{attribute 'qualified_only'}
{attribute 'strict'}
{attribute 'to_string'}
TYPE E_Alarm :
(
	AL000,
	AL001,
	AL002,
	AL003,
	AL004,
	AL005,
	AL006,
	AL007,
	AL008,
	AL009,
	AL010,
	AL011,
	AL012,
	AL013,
	AL014,
	AL015,
	AL016,
	AL017,
	AL018,
	AL019,
	AL020,
	AL021,
	AL022,
	AL023,
	AL024,
	AL025,
	AL026,
	AL027,
	AL028,
	AL029,
	AL030,
	AL031,
	AL032,
	AL033,
	AL034,
	AL035,
	AL036,
	AL037,
	AL038,
	AL039,
	AL040,
	AL041,
	AL042,
	AL043,
	AL044,
	AL045,
	AL046,
	AL047,
	AL048,
	AL049,
	AL050,
	AL051,
	AL052,
	AL053,
	AL054,
	AL055,
	AL056,
	AL057,
	AL058,
	AL059,
	AL060,
	AL061,
	AL062,
	AL063,
	AL064,
	AL065,
	AL066,
	AL067,
	AL068,
	AL069,
	AL070,
	AL071,
	AL072,
	AL073,
	AL074,
	AL075,
	AL076,
	AL077,
	AL078,
	AL079,
	AL080,
	AL081,
	AL082,
	AL083,
	AL084,
	AL085,
	AL086,
	AL087,
	AL088,
	AL089,
	AL090,
	AL091,
	AL092,
	AL093,
	AL094,
	AL095,
	AL096,
	AL097,
	AL098,
	AL099,
	AL100,
	AL101,
	AL102,
	AL103,
	AL104,
	AL105,
	AL106,
	AL107,
	AL108,
	AL109,
	AL110,
	AL111,
	AL112,
	AL113,
	AL114,
	AL115,
	AL116,
	AL117,
	AL118,
	AL119,
	AL120,
	AL121,
	AL122,
	AL123,
	AL124,
	AL125,
	AL126,
	AL127,
	AL128,
	AL129,
	AL130,
	AL131,
	AL132,
	AL133,
	AL134,
	AL135,
	AL136,
	AL137,
	AL138,
	AL139,
	AL140,
	AL141,
	AL142,
	AL143,
	AL144,
	AL145,
	AL146,
	AL147,
	AL148,
	AL149,
	AL150,
	AL151,
	AL152,
	AL153,
	AL154,
	AL155,
	AL156,
	AL157,
	AL158,
	AL159,
	AL160,
	AL161,
	AL162,
	AL163,
	AL164,
	AL165,
	AL166,
	AL167,
	AL168,
	AL169,
	AL170,
	AL171,
	AL172,
	AL173,
	AL174,
	AL175,
	AL176,
	AL177,
	AL178,
	AL179,
	AL180,
	AL181,
	AL182,
	AL183,
	AL184,
	AL185,
	AL186,
	AL187,
	AL188,
	AL189,
	AL190,
	AL191,
	AL192,
	AL193,
	AL194,
	AL195,
	AL196,
	AL197,
	AL198,
	AL199,
	AL200,
	AL201,
	AL202,
	AL203,
	AL204,
	AL205,
	AL206,
	AL207,
	AL208,
	AL209,
	AL210,
	AL211,
	AL212,
	AL213,
	AL214,
	AL215,
	AL216,
	AL217,
	AL218,
	AL219,
	AL220,
	AL221,
	AL222,
	AL223,
	AL224,
	AL225,
	AL226,
	AL227,
	AL228,
	AL229,
	AL230,
	AL231,
	AL232,
	AL233,
	AL234,
	AL235,
	AL236,
	AL237,
	AL238,
	AL239,
	AL240,
	AL241,
	AL242,
	AL243,
	AL244,
	AL245,
	AL246,
	AL247,
	AL248,
	AL249,
	AL250,
	AL251,
	AL252,
	AL253,
	AL254,
	AL255,
	AL256,
	AL257,
	AL258,
	AL259,
	AL260,
	AL261,
	AL262,
	AL263,
	AL264,
	AL265,
	AL266,
	AL267,
	AL268,
	AL269,
	AL270,
	AL271,
	AL272,
	AL273,
	AL274,
	AL275,
	AL276,
	AL277,
	AL278,
	AL279,
	AL280,
	AL281,
	AL282,
	AL283,
	AL284,
	AL285,
	AL286,
	AL287,
	AL288,
	AL289,
	AL290,
	AL291,
	AL292,
	AL293,
	AL294,
	AL295,
	AL296,
	AL297,
	AL298,
	AL299,
	AL300,
	AL301,
	AL302,
	AL303,
	AL304,
	AL305,
	AL306,
	AL307,
	AL308,
	AL309,
	AL310,
	AL311,
	AL312,
	AL313,
	AL314,
	AL315,
	AL316,
	AL317,
	AL318,
	AL319,
	AL320,
	AL321,
	AL322,
	AL323,
	AL324,
	AL325,
	AL326,
	AL327,
	AL328,
	AL329,
	AL330,
	AL331,
	AL332,
	AL333,
	AL334,
	AL335,
	AL336,
	AL337,
	AL338,
	AL339,
	AL340,
	AL341,
	AL342,
	AL343,
	AL344,
	AL345,
	AL346,
	AL347,
	AL348,
	AL349,
	AL350,
	AL351,
	AL352,
	AL353,
	AL354,
	AL355,
	AL356,
	AL357,
	AL358,
	AL359,
	AL360,
	AL361,
	AL362,
	AL363,
	AL364,
	AL365,
	AL366,
	AL367,
	AL368,
	AL369,
	AL370,
	AL371,
	AL372,
	AL373,
	AL374,
	AL375,
	AL376,
	AL377,
	AL378,
	AL379,
	AL380,
	AL381,
	AL382,  
	AL383,
	AL384,
	AL385,
	AL386,
	AL387,
	AL388,
	AL389,  
	AL390,
	AL391,
	AL392,
	AL393,
	AL394,
	AL395,
	AL396,
	AL397,
	AL398,
	AL399,
	AL400,//B槽主軸伺服馬達_軸錯誤異常   
	AL401,//B槽清洗內罩升降1馬達_軸錯誤異常
	AL402,//B槽清洗內罩升降2馬達_軸錯誤異常
	AL403,//B槽清洗外罩升降1馬達_軸錯誤異常
	AL404,//B槽清洗外罩升降2馬達_軸錯誤異常
	AL405,//B槽噴頭擺臂升降馬達_軸錯誤異常 
	AL406,//B槽噴頭擺臂馬達_軸錯誤異常   
	AL407,//B槽頂PIN升降馬達_軸錯誤異常
	AL408,//B槽噴頭X軸馬達_軸錯誤異常   
	AL409,//B槽噴頭Y1軸馬達_軸錯誤異常  
	AL410,//B槽噴頭Y2軸馬達_軸錯誤異常  
	AL411,//B槽噴頭Z軸馬達_軸錯誤異常
	AL412,//B槽噴頭T軸馬達_軸錯誤異常 
	AL413,//B槽主軸伺服馬達_驅動器異常   
	AL414,//B槽清洗內罩升降1馬達_驅動器異常
	AL415,//B槽清洗內罩升降2馬達_驅動器異常
	AL416,//B槽清洗外罩升降1馬達_驅動器異常
	AL417,//B槽清洗外罩升降2馬達_驅動器異常
	AL418,//B槽噴頭擺臂升降馬達_驅動器異常 
	AL419,//B槽噴頭擺臂馬達_驅動器異常   
	AL420,//B槽頂PIN升降馬達_驅動器異常 
	AL421,//B槽噴頭X軸馬達_驅動器異常   
	AL422,//B槽噴頭Y1軸馬達_驅動器異常  
	AL423,//B槽噴頭Y2軸馬達_驅動器異常  
	AL424,//B槽噴頭Z軸馬達_驅動器異常   
	AL425,//B槽噴頭T軸馬達_驅動器異常   
	AL426,//                 
	AL427,//                 
	AL428,//                 
	AL429,//                 
	AL430,//清洗內罩升降1到位檢知異常    
	AL431,//清洗內罩升降2到位檢知異常    
	AL432,//清洗外罩升降1到位檢知異常    
	AL433,//清洗外罩升降2到位檢知異常    
	AL434,//噴頭X軸到位檢知異常       
	AL435,//噴頭Z軸到位檢知異常       
	AL436,//噴頭Y1軸到位檢知異常      
	AL437,//噴頭Y2軸到位檢知異常      
	AL438,//頂PIN升降到位檢知異常     
	AL439,//噴頭擺臂升降到位檢知異常     
	AL440,//噴頭擺臂擺動到位檢知異常     
	AL441,//閘門磁簧開關1(關)異常     
	AL442,//閘門磁簧開關1(開)異常     
	AL443,//閘門磁簧開關2(關)異常     
	AL444,//閘門磁簧開關2(開)異常     
	AL445,//上擺臂定位汽缸磁簧開關(定位)異常
	AL446,//上擺臂定位汽缸磁簧開關(退)異常 
	AL447,//下擺臂定位汽缸磁簧開關(定位)異常
	AL448,//下擺臂定位汽缸磁簧開關(退)異常 
	AL449,//上擺臂切換光電素子異常      
	AL450,//下擺臂切換光電素子異常      
	AL451,//DIW混CO2加熱器EGO異常  
	AL452,//DIW加熱器EGO異常      
	AL453,//漏液檢知器異常          
	AL454,//                 
	AL455,//                 
	AL456,//                 
	AL457,//                 
	AL458,//                 
	AL459,//                 
	AL460,//                 
	AL461,//                 
	AL462,//                 
	AL463,//                 
	AL464,//                 
	AL465,//                 
	AL466,//                 
	AL467,//                 
	AL468,//                 
	AL469,//                 
	AL470,//                 
	AL471,//                 
	AL472,//                 
	AL473,//                 
	AL474,//                 
	AL475,//                 
	AL476,//                 
	AL477,//                 
	AL478,//                 
	AL479,//                 
	AL480,//                 
	AL481,//                 
	AL482,//                 
	AL483,//                 
	AL484,//                 
	AL485,//                 
	AL486,//                 
	AL487,//                 
	AL488,//                 
	AL489,//                 
	AL490,//                 
	AL491,//                 
	AL492,//                 
	AL493,//                 
	AL494,//                 
	AL495,//                 
	AL496,//                 
	AL497,//                 
	AL498,//                 
	AL499,//                 
	AL500,//                 
	AL501,//                 
	AL502,//                 
	AL503,//                 
	AL504,//                 
	AL505,//                 
	AL506,//                 
	AL507,//                 
	AL508,//                 
	AL509,//                 
	AL510,//                 
	AL511,//                 
	AL512,//                 
	AL513,//                 
	AL514,//                 
	AL515,//                 
	AL516,//                 
	AL517,//                 
	AL518,//                 
	AL519,//                 
	AL520,//                 
	AL521,//                 
	AL522,//                 
	AL523,//                 
	AL524,//                 
	AL525,//                 
	AL526,//                 
	AL527,//                 
	AL528,//                 
	AL529,//                 
	AL530,//                 
	AL531,//                 
	AL532,//                 
	AL533,//                 
	AL534,//                 
	AL535,//                 
	AL536,//                 
	AL537,//                 
	AL538,//                 
	AL539,//                 
	AL540,//                 
	AL541,//                 
	AL542,//                 
	AL543,//                 
	AL544,//                 
	AL545,//                 
	AL546,//                 
	AL547,//                 
	AL548,//                 
	AL549,//                 
	AL550,//                 
	AL551,//                 
	AL552,//                 
	AL553,//                 
	AL554,//                 
	AL555,//                 
	AL556,//                 
	AL557,//                 
	AL558,//                 
	AL559,//                 
	AL560,//                 
	AL561,//                 
	AL562,//                 
	AL563,//                 
	AL564,//                 
	AL565,//                 
	AL566,//                 
	AL567,//                 
	AL568,//                 
	AL569,//                 
	AL570,//                 
	AL571,//                 
	AL572,//                 
	AL573,//                 
	AL574,//                 
	AL575,//                 
	AL576,//                 
	AL577,//                 
	AL578,//                 
	AL579,//                 
	AL580,//                 
	AL581,//                 
	AL582,//                 
	AL583,//                 
	AL584,//                 
	AL585,//                 
	AL586,//                 
	AL587,//                 
	AL588,//                 
	AL589,//                 
	AL590,//                 
	AL591,//                 
	AL592,//                 
	AL593,//                 
	AL594,//                 
	AL595,//                 
	AL596,//                 
	AL597,//                 
	AL598,//                 
	AL599 //                 
);
END_TYPE

(* stored: Version 1.1.0.1, ProductVersion 3.1.4026.18
   DUT E_Alarm: Id {895b1ec5-7ade-44d3-a317-bca7ecd292a0} *)
